FUNCTION F_TargetWindowReached : BOOL
VAR_INPUT
	fCurrentPos: LREAL;
	fTargetPos: LREAL;
	fWindow: LREAL;
END_VAR


F_TargetWindowReached := fCurrentPos >= (fTargetPos - fWindow) AND fCurrentPos <= (fTargetPos + fWindow);

END_FUNCTION

(* stored: Version 1.1.0.1, ProductVersion 3.1.4022.9
   POU F_TargetWindowReached: Id {293b00b7-c73e-4ece-9e85-9140e5ea5bc9}, SpecialFunc None *)
